TYPE stCMD_SET :
STRUCT
	command_for_battery: REAL;
	plant_sp: REAL;
END_STRUCT
END_TYPE

(* stored: Version 1.1.0.1, ProductVersion 3.1.4026.11
   DUT stCMD_SET: Id {0524fe45-0c39-4c6a-983a-b5f5fc4ea561} *)
